RoboDK station: RoboDK sw01 UR3e-first Test with real Robot.rdk

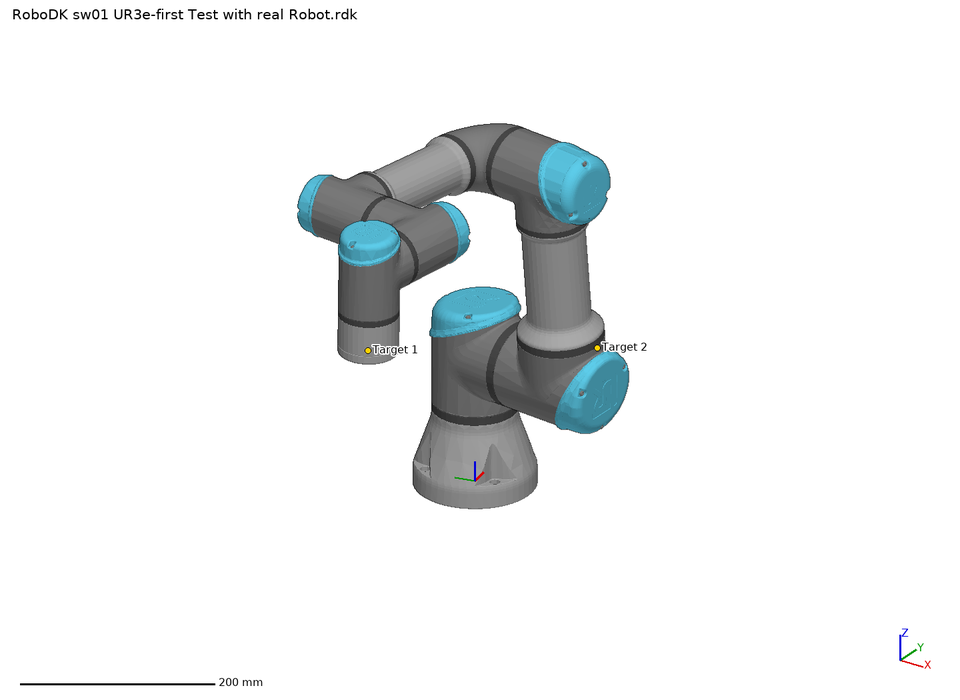
[picture v0: the station drawn from its stored meshes, robots at their saved joint values, targets as dots, program paths as lines]
Station RoboDK sw01 UR3e-first Test with real Robot (saved by RoboDK 5.9.5). Poses are relative to the parent item; angles as X-Y-Z fixed-axis rotations.
  - frame UR3e Base at (0, 0, 0) mm, rotated rx 0 ry 0 rz 101.86 deg
    - robot UR3e: 6 axes, payload 3 kg, reach 500 mm, repeatability 0.03 mm, weight 11 kg
        modified DH rows (alpha deg, a mm, theta deg, d mm): 0, 0, 0, 151.9; 90, 0, 180, 0; 0, 243.55, 0, 0; 0, 213.2, 0, 131.05; -90, 0, 0, 85.35; 90, 0, 180, 92.1
        joint limits [-360, -360, -360, -360, -360, -360] to [360, 360, 360, 360, 360, 360]; home [0, -90, -90, 0, 90, 0]; saved at [-17.216, -84.463, 82.469, -87.777, -90.911, -268.656]
  - frame UR3e Base at (0, 1000, 0) mm
    - target Target 1 (Cartesian target) at (98.79, -1332.3, 309.29) mm, rotated rx -179.09 ry -0.21 rz 83.26 deg; joints [84.606, -84.464, 82.472, -87.774, -90.909, -268.658] of UR3e
    - target Target 2 (Cartesian target) at (288.12, -1192.79, 309.29) mm, rotated rx -179.09 ry -0.21 rz 122.92 deg; joints [22.398, -84.464, 82.472, -87.774, -90.909, -268.658] of UR3e
